PROGRAM kleurmachine
VAR
	state : KleurmachineToestand;
	
	
	kleurmachineReady : BOOL;
	kleurmachineBezig : BOOL;
	
	inputCode : INT;
	goedeCode : INT := 1234;
	
	kleurmachineTimer : TON;
END_VAR

CASE state OF
	KleurmachineToestand.startup:
		// Simulate startup
		kleurmachineTimer(IN:=TRUE, PT:=T#10S);
		IF kleurmachineTimer.Q THEN
			kleurmachineTimer(IN:=FALSE);
			state := KleurmachineToestand.home;
		END_IF
		
	KleurmachineToestand.home:
		kleurmachineReady := TRUE;
		kleurmachineBezig := FALSE;
		IF GVL.opdrachtKnop THEN
			state := KleurmachineToestand.info;
		END_IF
		
	KleurmachineToestand.info:
		IF GVL.startKnop THEN
			state := KleurmachineToestand.scan;
		END_IF
		
	KleurmachineToestand.scan:
		kleurmachineReady := FALSE;
		kleurmachineBezig := TRUE;
		IF GVL.barcodeBlik = goedeCode THEN
			state := KleurmachineToestand.wachtOpBlik;
		END_IF
		
	KleurmachineToestand.wachtOpBlik:
		IF GVL.blikPresent OR GVL.okeKnop THEN
			state := KleurmachineToestand.kleurToevoegen;
		END_IF
		
	KleurmachineToestand.kleurToevoegen:
		IF GVL.verfOrder[4] = '2.5' THEN
			kleurmachineTimer(IN:=TRUE,PT:=T#20S); // simulate the colors being added
		ELSIF GVL.verfOrder[4] = '5' THEN
			kleurmachineTimer(IN:=TRUE,PT:=T#30S); // simulate the colors being added
		ELSIF GVL.verfOrder[4] = '10' THEN
			kleurmachineTimer(IN:=TRUE,PT:=T#40S); // simulate the colors being added
		END_IF
		
		IF kleurmachineTimer.Q THEN
			state := KleurmachineToestand.klaarMetToevoegen;
		END_IF
		
	KleurmachineToestand.klaarMetToevoegen:
		IF GVL.okeKnop OR NOT GVL.blikPresent THEN
			state := KleurmachineToestand.home;	
		END_IF
END_CASE

END_PROGRAM

(* stored: Version 1.1.0.1, ProductVersion 3.1.4024.15
   POU kleurmachine: Id {e2f2c538-0dc9-411e-a330-8428cfac9392}, SpecialFunc None *)
